Fanuc KAREL source: kd00025.KL

-- PROVISIONAL review KL for V770-1; original PC SHA256 01196057baaf17891af60a0c047380441c18aa0d516a5df1b12b6a8cd51c0bad
-- Incomplete behavior may be omitted. Consult companion uncertainty JSON. Do not deploy.
PROGRAM KD00025
%NOLOCKGROUP
VAR
  I : INTEGER
  J : INTEGER
  B : BOOLEAN
  R : REAL
  S : STRING[80]
BEGIN
  -- UNRESOLVED_PC offsets 5-31; opcodes 9D,2E,25,81,18,9D,1B,9D,12,22,9D,13,04
  -- UNRESOLVED_PC offsets 36-40; opcodes 7F
END KD00025
